Staubli VAL3: onF7Event.pgx

program onF7Event(bool& x_bSave[])
  local string l_sMessage
  local bool l_bFound
  local string l_sTrajName
  local bool l_bYes
  local string l_sString
  local string l_sButton[2]
begin
  // look if the bButton is enable
  if bButton[6]
    // delete the selected tool
    if  nIndexTool!=0
      call language:message(l_sMessage,120)
      // get the yes_no button
      call language:getYesNo(l_sButton)
      // ask the question
      call use:yes_no(l_sMessage+toString("",nIndexTool),l_sButton,l_bYes)
      if l_bYes
        call refreshStatic()

        if !l_bFound
          // move from the all traj the indexTool

          call tcp:delete(nIndexTool)
          nIndexTool=nIndexTool-1
          logMsg("[VALlaser] INTERFACE:Delete the tool: "+toString("",nIndexTool))
          x_bSave=true
        else
          // show the message the tool is already used
          call language:message(l_sMessage,124)
          call language:message(l_sString,29)
          popUpMsg(l_sMessage+l_sString+l_sTrajName)
        endIf
      endIf
    endIf
  endIf
end
